(* IEC 61131-3 sources: ics/BLR1_PhoenixContact/BLR1_AXC1050_21/LogicalPOUs/MB, 7 files *)

(* ---- DW_TO_DWORD.ST ---- *)
(*@PROPERTIES_EX@
TYPE: POU
LOCALE: 0
IEC_LANGUAGE: ST
PLC_TYPE: independent
PROC_TYPE: independent
GROUP: MB.FB
*)
(*@KEY@:DESCRIPTION*)

(*@KEY@:END_DESCRIPTION*)
FUNCTION DW_TO_DWORD:DWORD

(*Group:Default*)

VAR_INPUT
    LO_WORD :	WORD;
    HI_WORD :	WORD;
END_VAR

VAR
    OUT_DWORD :	DWORD;
END_VAR

(*@KEY@: WORKSHEET
NAME: DW_TO_DWORD
IEC_LANGUAGE: ST
*)
OUT_DWORD.W0:=HI_WORD;
OUT_DWORD.W1:=LO_WORD;
DW_TO_DWORD:=OUT_DWORD;

(*@KEY@: END_WORKSHEET *)
END_FUNCTION

(* ---- MB_TO_REAL.ST ---- *)
(*@PROPERTIES_EX@
TYPE: POU
LOCALE: 0
IEC_LANGUAGE: ST
PLC_TYPE: independent
PROC_TYPE: independent
GROUP: MB.FB
*)
(*@KEY@:DESCRIPTION*)

(*@KEY@:END_DESCRIPTION*)
FUNCTION_BLOCK MB_TO_REAL

(*Group:Default*)

VAR_INPUT
	LoWord :	WORD;
	HiWord :	WORD;
END_VAR

VAR
	SYS_IEEE_ToReal_1_1 :	SYS_IEEE_ToReal_1;
END_VAR

VAR_OUTPUT
	OUT :	REAL;
END_VAR

VAR
	IEEE :	SYS_ARR_B_1_4;
END_VAR

(*@KEY@: WORKSHEET
NAME: MB_TO_REAL
IEC_LANGUAGE: ST
*)

IEEE[1]:= LoWord.B0;
IEEE[2]:= LoWord.B1;
IEEE[3]:= HiWord.B0;
IEEE[4]:= HiWord.B1;

SYS_IEEE_ToReal_1_1(arrIEEE_Float:= IEEE);
OUT:=SYS_IEEE_ToReal_1_1.rValue;

(*@KEY@: END_WORKSHEET *)
END_FUNCTION_BLOCK

(* ---- MB_TO_REAL_1.ST ---- *)
(*@PROPERTIES_EX@
TYPE: POU
LOCALE: 0
IEC_LANGUAGE: ST
PLC_TYPE: independent
PROC_TYPE: independent
GROUP: MB.FB
*)
(*@KEY@:DESCRIPTION*)

(*@KEY@:END_DESCRIPTION*)
FUNCTION_BLOCK MB_TO_REAL_1

(*Group:Default*)

VAR_INPUT
	LoWord :	WORD;
	HiWord :	WORD;
END_VAR

VAR
	SYS_IEEE_ToReal_1_1 :	SYS_IEEE_ToReal_1;
END_VAR

VAR_OUTPUT
	OUT :	REAL;
END_VAR

VAR
	IEEE :	SYS_ARR_B_1_4;
END_VAR

(*@KEY@: WORKSHEET
NAME: MB_TO_REAL_1
IEC_LANGUAGE: ST
*)

IEEE[1]:= LoWord.B1;
IEEE[2]:= LoWord.B0;
IEEE[3]:= HiWord.B1;
IEEE[4]:= HiWord.B0;

SYS_IEEE_ToReal_1_1(arrIEEE_Float:= IEEE);
OUT:=SYS_IEEE_ToReal_1_1.rValue;

(*@KEY@: END_WORKSHEET *)
END_FUNCTION_BLOCK

(* ---- REAL_TO_MB.ST ---- *)
(*@PROPERTIES_EX@
TYPE: POU
LOCALE: 0
IEC_LANGUAGE: ST
PLC_TYPE: independent
PROC_TYPE: independent
GROUP: MB.FB
*)
(*@KEY@:DESCRIPTION*)

(*@KEY@:END_DESCRIPTION*)
FUNCTION_BLOCK REAL_TO_MB

(*Group:Default*)

VAR_OUTPUT
	LoWord :	WORD;
	HiWord :	WORD;
END_VAR

VAR_INPUT
	IN :	REAL;
END_VAR

VAR
	SYS_RealTo_IEEE_1_1 :	SYS_RealTo_IEEE_1;
	IEEE :	SYS_ARR_B_1_4;
END_VAR

(*@KEY@: WORKSHEET
NAME: REAL_TO_MB
IEC_LANGUAGE: ST
*)

SYS_RealTo_IEEE_1_1(rValue:=IN);
IEEE:=SYS_RealTo_IEEE_1_1.arrIEEE_Float;

LoWord.B0:= IEEE[1];
LoWord.B1:= IEEE[2];
HiWord.B0:= IEEE[3];
HiWord.B1:= IEEE[4];
(*@KEY@: END_WORKSHEET *)
END_FUNCTION_BLOCK

(* ---- MB_RTU_1.ST ---- *)
(*@PROPERTIES_EX@
TYPE: POU
LOCALE: 0
IEC_LANGUAGE: ST
PLC_TYPE: independent
PROC_TYPE: independent
GROUP: MB
*)
(*@KEY@:DESCRIPTION*)

(*@KEY@:END_DESCRIPTION*)
PROGRAM MB_RTU_1

(*Group:NewGroup*)

VAR
    TON_MB_RTU_Master_Startup :	TON;
    MB_AXL_RS_UNI_Act :	BOOL;
    MB_RTU_Master_Act :	BOOL;
    MB_RTU_FC_Act :	BOOL;
    MB_AXL_RS_UNI_REC_2_1 :	MB_AXL_RS_UNI_REC_2;
    udtSerialIF :	MB2_AXL_RSUNI2_UDT_IF;
END_VAR

VAR_EXTERNAL
    arrInData_AXL_RSUNI_1 :	MB2_AXL_RSUNI2_ARR_B_0_19;
    arrOutData_AXL_RSUNI_1 :	MB2_AXL_RSUNI2_ARR_B_0_19;
END_VAR

VAR
    udtDiag_AXL_RSUNI_REC :	MB_UDT_RTU_REC_DIAG;
    wDiagCode_AXL_RSUNI_REC :	WORD;
    wAddDiagCode_AXL_RSUNI_REC :	WORD;
    xError_AXL_RSUNI_REC :	BOOL;
    xBusy_AXL_RSUNI_REC :	BOOL;
    xActive_AXL_RSUNI_REC :	BOOL;
    MB_AXL_RS_UNI_SND_2_1 :	MB_AXL_RS_UNI_SND_2;
    udtDiag_AXL_RSUNI_SND :	MB_UDT_RTU_SND_DIAG;
    wAddDiagCode_AXL_RSUNI_SND :	WORD;
    wDiagCode_AXL_RSUNI_SND :	WORD;
    xError_AXL_RSUNI_SND :	BOOL;
    xBusy_AXL_RSUNI_SND :	BOOL;
    xActive_AXL_RSUNI_SND :	BOOL;
    MB_RTU_Master_4_1 :	MB_RTU_Master_4;
    udtMbData :	udtModbus2_Data;
    udtDiag_RTU_Master :	MB_UDT_RTU_MASTER_DIAG;
    wAddDiagCode_RTU_Master :	WORD;
    wDiagCode_RTU_Master :	WORD;
    xError_RTU_Master :	BOOL;
    xBusy_RTU_Master :	BOOL;
    xActive_RTU_Master :	BOOL;
    uiRespCount_RTU_Master :	UINT;
    uiReqCount_RTU_Master :	UINT;
    MB_RTU_FC3 :	MB_RTU_FC3_3;
    SlvAddr :	MBRTU_SlvAddr;
    RegAddr :	MBRTU_RegAddr;
    arrReadData_RTU_FC3 :	arrModbus2_W_1_125;
    udtDiag_RTU_FC3 :	MB_UDT_RTU_FC_DIAG;
    wAddDiagCode_RTU_FC3 :	WORD;
    wDiagCode_RTU_FC3 :	WORD;
    xError_RTU_FC3 :	BOOL;
    xDone_RTU_FC3 :	BOOL;
    xBusy_RTU_FC3 :	BOOL;
    xActive_RTU_FC3 :	BOOL;
    R_TRIG_1 :	R_TRIG;
    F_TRIG_3 :	F_TRIG;
    i :	INT;
    j :	INT;
    a :	INT;
    b :	INT;
    i1 :	INT;
    State :	INT;
    xSndReq_RTU_FC3 :	BOOL;
END_VAR

VAR_EXTERNAL
    SlvData_RSUNI_1 :	MBRTU_SlvData;
    PLCMODE_RUN :	BOOL;(*PLC status RUN*)
END_VAR

(*@KEY@: WORKSHEET
NAME: MB_RTU_1
IEC_LANGUAGE: ST
*)
(*============================================================================*)
(*MB RTU startup timer*)
(*============================================================================*)
TON_MB_RTU_Master_Startup(IN:= PLCMODE_RUN,PT:=t#2s);
IF TON_MB_RTU_Master_Startup.Q and not (xError_AXL_RSUNI_REC or
    xError_RTU_Master or xError_AXL_RSUNI_SND) THEN
    MB_AXL_RS_UNI_Act		:= true;
    MB_RTU_Master_Act		:= true;
    MB_RTU_FC_Act			:= true;
ELSE
    MB_AXL_RS_UNI_Act		:= false;
    MB_RTU_Master_Act		:= false;
    MB_RTU_FC_Act			:= false;
END_IF;

(*============================================================================*)
(*MB_AXL_UNI_REC FB initialization*)
(*============================================================================*)
MB_AXL_RS_UNI_REC_2_1(xActivate:= MB_AXL_RS_UNI_Act,
    udtSerialIF:= udtSerialIF,
    arrInputData:= arrInData_AXL_RSUNI_1,
    arrOutputData:= arrOutData_AXL_RSUNI_1);

xActive_AXL_RSUNI_REC		:=MB_AXL_RS_UNI_REC_2_1.xActive;
xBusy_AXL_RSUNI_REC			:=MB_AXL_RS_UNI_REC_2_1.xBusy;
xError_AXL_RSUNI_REC		:=MB_AXL_RS_UNI_REC_2_1.xError;
wDiagCode_AXL_RSUNI_REC		:=MB_AXL_RS_UNI_REC_2_1.wDiagCode;
wAddDiagCode_AXL_RSUNI_REC	:=MB_AXL_RS_UNI_REC_2_1.wAddDiagCode;
udtDiag_AXL_RSUNI_REC		:=MB_AXL_RS_UNI_REC_2_1.udtDiag;
udtSerialIF					:=MB_AXL_RS_UNI_REC_2_1.udtSerialIF;
arrInData_AXL_RSUNI_1		:=MB_AXL_RS_UNI_REC_2_1.arrInputData;
arrOutData_AXL_RSUNI_1		:=MB_AXL_RS_UNI_REC_2_1.arrOutputData;

(*============================================================================*)
(*MB RTU Master FB initialization*)
(*============================================================================*)
MB_RTU_Master_4_1(xActivate:= xActive_AXL_RSUNI_REC and xActive_AXL_RSUNI_SND,
    xReset:= false,
    xAuto_CRC:= false,
    tTimeout:= t#200ms,
    udtSerialIF:= udtSerialIF,
    udtMbData:= udtMbData);

xActive_RTU_Master			:=MB_RTU_Master_4_1.xActive;
xBusy_RTU_Master			:=MB_RTU_Master_4_1.xBusy;
uiReqCount_RTU_Master		:=MB_RTU_Master_4_1.uiRequestsCounter;
uiRespCount_RTU_Master		:=MB_RTU_Master_4_1.uiResponsesCounter;
xError_RTU_Master			:=MB_RTU_Master_4_1.xError;
wDiagCode_RTU_Master		:=MB_RTU_Master_4_1.wDiagCode;
wAddDiagCode_RTU_Master		:=MB_RTU_Master_4_1.wAddDiagCode;
udtDiag_RTU_Master			:=MB_RTU_Master_4_1.udtDiag;
udtSerialIF					:=MB_RTU_Master_4_1.udtSerialIF;
udtMbData					:=MB_RTU_Master_4_1.udtMbData;

(*============================================================================*)
(*MB_AXL_UNI_SND FB initialization*)
(*============================================================================*)
MB_AXL_RS_UNI_SND_2_1(xActivate:= MB_AXL_RS_UNI_Act,
    udtSerialIF:= udtSerialIF,
    arrInputData:= arrInData_AXL_RSUNI_1,
    arrOutputData:= arrOutData_AXL_RSUNI_1);

xActive_AXL_RSUNI_SND		:=MB_AXL_RS_UNI_SND_2_1.xActive;
xBusy_AXL_RSUNI_SND			:=MB_AXL_RS_UNI_SND_2_1.xBusy;
xError_AXL_RSUNI_SND		:=MB_AXL_RS_UNI_SND_2_1.xError;
wDiagCode_AXL_RSUNI_SND		:=MB_AXL_RS_UNI_SND_2_1.wDiagCode;
wAddDiagCode_AXL_RSUNI_SND	:=MB_AXL_RS_UNI_SND_2_1.wAddDiagCode;
udtDiag_AXL_RSUNI_SND		:=MB_AXL_RS_UNI_SND_2_1.udtDiag;
udtSerialIF					:=MB_AXL_RS_UNI_SND_2_1.udtSerialIF;
arrInData_AXL_RSUNI_1		:=MB_AXL_RS_UNI_SND_2_1.arrInputData;
arrOutData_AXL_RSUNI_1		:=MB_AXL_RS_UNI_SND_2_1.arrOutputData;

(*============================================================================*)
(*Slaves registers addresses assigning*)
(*============================================================================*)
R_TRIG_1(CLK:= xActive_RTU_Master);

SlvAddr[0]					:= uint#10;                                         (*Pump 5.1 FC MB address*)
SlvAddr[1]					:= uint#11;                                         (*Pump 5.2 FC MB address*)
SlvAddr[2]					:= uint#12;                                         (*Pump 5.3 FC MB address*)

IF R_TRIG_1.Q THEN
    i:= 0;
    j:= 0;
    FOR i1:= 0 to 2 DO
        RegAddr[i1][0]		:= uint#16129;                                      (*reg.16129 Frequency Hz*)
        RegAddr[i1][1]		:= uint#16099;                                      (*reg.16099 Power kWt*)
        RegAddr[i1][2]		:= uint#16139;                                      (*reg.16139 Motor Current A*)
        RegAddr[i1][3]		:= uint#16339;                                      (*reg.16339 HeatSink Temp.*)
        RegAddr[i1][4]		:= uint#16029;                                      (*reg.16029 Status Word*)
        RegAddr[i1][5]		:= uint#16899;                                      (*reg.16899 Alarm Word*)
        RegAddr[i1][6]		:= uint#16919;                                      (*reg.16919 Warning Word*)
        RegAddr[i1][7]		:= uint#15009;                                      (*reg.15009 Running hours h*)
        RegAddr[i1][8]		:= uint#15019;                                      (*reg.15019 kWh Counter*)
    END_FOR;
END_IF;

(*============================================================================*)
(*Pumps FCs parameters reading*)
(*============================================================================*)
MB_RTU_FC3(xActivate:= MB_RTU_Master_Act,
    xSendRequest:= xSndReq_RTU_FC3,
    xEnablePoll:= false,
    tPollInterval:= t#100ms,
    uiSlaveAddress:= SlvAddr[i],
    uiStartAddress:=RegAddr[i][j],
    iDataCount:= 2,
    arrReadData:= arrReadData_RTU_FC3,
    udtMbData:= udtMbData);

xActive_RTU_FC3				:=MB_RTU_FC3.xActive;
xBusy_RTU_FC3				:=MB_RTU_FC3.xBusy;
xDone_RTU_FC3				:=MB_RTU_FC3.xDone;
xError_RTU_FC3				:=MB_RTU_FC3.xError;
wDiagCode_RTU_FC3			:=MB_RTU_FC3.wDiagCode;
wAddDiagCode_RTU_FC3		:=MB_RTU_FC3.wAddDiagCode;
udtDiag_RTU_FC3				:=MB_RTU_FC3.udtDiag;
arrReadData_RTU_FC3			:=MB_RTU_FC3.arrReadData;
udtMbData					:=MB_RTU_FC3.udtMbData;

CASE State OF
    0:
        IF xActive_RTU_Master THEN
            xSndReq_RTU_FC3 := true;
            State:= 10;
        END_IF;

    10:
        IF MB_RTU_FC3.xDone or MB_RTU_FC3.xError THEN
            xSndReq_RTU_FC3 := false;
            State:= 100;
        END_IF;

    100:
        a:= j * 2;
        b:= a + 1;

        SlvData_RSUNI_1[i][a]:= arrReadData_RTU_FC3[1];
        SlvData_RSUNI_1[i][b]:= arrReadData_RTU_FC3[2];
        State:= 1000;

    1000:
        j:= j + 1;
        IF j > 8 THEN
            j:= 0;
            i:= i + 1;
        END_IF;

        IF i > 2 THEN
            i:= 0;
        END_IF;

        State:= 0;
END_CASE;

(*@KEY@: END_WORKSHEET *)
END_PROGRAM

(* ---- MB_RTU_2.ST ---- *)
(*@PROPERTIES_EX@
TYPE: POU
LOCALE: 0
IEC_LANGUAGE: ST
PLC_TYPE: independent
PROC_TYPE: independent
GROUP: MB
*)
(*@KEY@:DESCRIPTION*)

(*@KEY@:END_DESCRIPTION*)
PROGRAM MB_RTU_2

(*Group:NewGroup*)

VAR
	TON_MB_RTU_Master_Startup :	TON;
	MB_AXL_RS_UNI_Act :	BOOL;
	MB_RTU_Master_Act :	BOOL;
	MB_RTU_FC_Act :	BOOL;
	MB_AXL_RS_UNI_REC_2_1 :	MB_AXL_RS_UNI_REC_2;
	udtSerialIF :	MB2_AXL_RSUNI2_UDT_IF;
END_VAR

VAR_EXTERNAL
	arrInData_AXL_RSUNI_2 :	MB2_AXL_RSUNI2_ARR_B_0_19;
	arrOutData_AXL_RSUNI_2 :	MB2_AXL_RSUNI2_ARR_B_0_19;
END_VAR

VAR
	udtDiag_AXL_RSUNI_REC :	MB_UDT_RTU_REC_DIAG;
	wDiagCode_AXL_RSUNI_REC :	WORD;
	wAddDiagCode_AXL_RSUNI_REC :	WORD;
	xError_AXL_RSUNI_REC :	BOOL;
	xBusy_AXL_RSUNI_REC :	BOOL;
	xActive_AXL_RSUNI_REC :	BOOL;
	MB_AXL_RS_UNI_SND_2_1 :	MB_AXL_RS_UNI_SND_2;
	udtDiag_AXL_RSUNI_SND :	MB_UDT_RTU_SND_DIAG;
	wAddDiagCode_AXL_RSUNI_SND :	WORD;
	wDiagCode_AXL_RSUNI_SND :	WORD;
	xError_AXL_RSUNI_SND :	BOOL;
	xBusy_AXL_RSUNI_SND :	BOOL;
	xActive_AXL_RSUNI_SND :	BOOL;
	MB_RTU_Master_4_1 :	MB_RTU_Master_4;
	udtMbData :	udtModbus2_Data;
	udtDiag_RTU_Master :	MB_UDT_RTU_MASTER_DIAG;
	wAddDiagCode_RTU_Master :	WORD;
	wDiagCode_RTU_Master :	WORD;
	xError_RTU_Master :	BOOL;
	xBusy_RTU_Master :	BOOL;
	xActive_RTU_Master :	BOOL;
	uiRespCount_RTU_Master :	UINT;
	uiReqCount_RTU_Master :	UINT;
	MB_RTU_FC3 :	MB_RTU_FC3_3;
	SlvAddr :	MBRTU_SlvAddr;
	RegAddr :	MBRTU_RegAddr;
	arrReadData_RTU_FC3 :	arrModbus2_W_1_125;
	udtDiag_RTU_FC3 :	MB_UDT_RTU_FC_DIAG;
	wAddDiagCode_RTU_FC3 :	WORD;
	wDiagCode_RTU_FC3 :	WORD;
	xError_RTU_FC3 :	BOOL;
	xDone_RTU_FC3 :	BOOL;
	xBusy_RTU_FC3 :	BOOL;
	xActive_RTU_FC3 :	BOOL;
	R_TRIG_1 :	R_TRIG;
	F_TRIG_3 :	F_TRIG;
	i :	INT;
	j :	INT;
	a :	INT;
	State :	INT;
	xSndReq_RTU_FC3 :	BOOL;
	b :	INT;
END_VAR

VAR_EXTERNAL
	SlvData_RSUNI_2 :	MBRTU_SlvData;
END_VAR

VAR
	i1 :	INT;
END_VAR

VAR_EXTERNAL
	PLCMODE_RUN :	BOOL;(*PLC status RUN*)
END_VAR

VAR
	FLG :	BOOL;
END_VAR

(*@KEY@: WORKSHEET
NAME: MB_RTU_2
IEC_LANGUAGE: ST
*)
(*============================================================================*)
(*MB RTU startup timer*)
(*============================================================================*)
TON_MB_RTU_Master_Startup(IN:=PLCMODE_RUN,PT:=t#2s);
IF TON_MB_RTU_Master_Startup.Q and not (xError_AXL_RSUNI_REC or xError_RTU_Master
	or xError_AXL_RSUNI_SND) THEN
	MB_AXL_RS_UNI_Act		:= true;
	MB_RTU_Master_Act		:= true;
	MB_RTU_FC_Act			:= true;
ELSE
	MB_AXL_RS_UNI_Act		:= false;
	MB_RTU_Master_Act		:= false;
	MB_RTU_FC_Act			:= false;
END_IF;

(*============================================================================*)
(*MB_AXL_UNI_REC FB initialization*)
(*============================================================================*)
MB_AXL_RS_UNI_REC_2_1(xActivate:= MB_AXL_RS_UNI_Act,
	udtSerialIF:= udtSerialIF,
	arrInputData:= arrInData_AXL_RSUNI_2,
	arrOutputData:= arrOutData_AXL_RSUNI_2);

xActive_AXL_RSUNI_REC		:=MB_AXL_RS_UNI_REC_2_1.xActive;
xBusy_AXL_RSUNI_REC			:=MB_AXL_RS_UNI_REC_2_1.xBusy;
xError_AXL_RSUNI_REC		:=MB_AXL_RS_UNI_REC_2_1.xError;
wDiagCode_AXL_RSUNI_REC		:=MB_AXL_RS_UNI_REC_2_1.wDiagCode;
wAddDiagCode_AXL_RSUNI_REC	:=MB_AXL_RS_UNI_REC_2_1.wAddDiagCode;
udtDiag_AXL_RSUNI_REC		:=MB_AXL_RS_UNI_REC_2_1.udtDiag;
udtSerialIF					:=MB_AXL_RS_UNI_REC_2_1.udtSerialIF;
arrInData_AXL_RSUNI_2		:=MB_AXL_RS_UNI_REC_2_1.arrInputData;
arrOutData_AXL_RSUNI_2		:=MB_AXL_RS_UNI_REC_2_1.arrOutputData;

(*============================================================================*)
(*MB RTU Master FB initialization*)
(*============================================================================*)
MB_RTU_Master_4_1(xActivate:= xActive_AXL_RSUNI_REC and xActive_AXL_RSUNI_SND,
	xReset:= false,
	xAuto_CRC:= false,
	tTimeout:= t#200ms,
	udtSerialIF:= udtSerialIF,
	udtMbData:= udtMbData);

xActive_RTU_Master			:=MB_RTU_Master_4_1.xActive;
xBusy_RTU_Master			:=MB_RTU_Master_4_1.xBusy;
uiReqCount_RTU_Master		:=MB_RTU_Master_4_1.uiRequestsCounter;
uiRespCount_RTU_Master		:=MB_RTU_Master_4_1.uiResponsesCounter;
xError_RTU_Master			:=MB_RTU_Master_4_1.xError;
wDiagCode_RTU_Master		:=MB_RTU_Master_4_1.wDiagCode;
wAddDiagCode_RTU_Master		:=MB_RTU_Master_4_1.wAddDiagCode;
udtDiag_RTU_Master			:=MB_RTU_Master_4_1.udtDiag;
udtSerialIF					:=MB_RTU_Master_4_1.udtSerialIF;
udtMbData					:=MB_RTU_Master_4_1.udtMbData;

(*============================================================================*)
(*MB_AXL_UNI_SND FB initialization*)
(*============================================================================*)
MB_AXL_RS_UNI_SND_2_1(xActivate:= MB_AXL_RS_UNI_Act,
	udtSerialIF:= udtSerialIF,
	arrInputData:= arrInData_AXL_RSUNI_2,
	arrOutputData:= arrOutData_AXL_RSUNI_2);

xActive_AXL_RSUNI_SND		:=MB_AXL_RS_UNI_SND_2_1.xActive;
xBusy_AXL_RSUNI_SND			:=MB_AXL_RS_UNI_SND_2_1.xBusy;
xError_AXL_RSUNI_SND		:=MB_AXL_RS_UNI_SND_2_1.xError;
wDiagCode_AXL_RSUNI_SND		:=MB_AXL_RS_UNI_SND_2_1.wDiagCode;
wAddDiagCode_AXL_RSUNI_SND	:=MB_AXL_RS_UNI_SND_2_1.wAddDiagCode;
udtDiag_AXL_RSUNI_SND		:=MB_AXL_RS_UNI_SND_2_1.udtDiag;
udtSerialIF					:=MB_AXL_RS_UNI_SND_2_1.udtSerialIF;
arrInData_AXL_RSUNI_2		:=MB_AXL_RS_UNI_SND_2_1.arrInputData;
arrOutData_AXL_RSUNI_2		:=MB_AXL_RS_UNI_SND_2_1.arrOutputData;

(*============================================================================*)
(*Slaves registers addresses assigning*)
(*============================================================================*)
R_TRIG_1(CLK:= xActive_RTU_Master);

SlvAddr[0]					:= uint#10;											(*Pump 3.1 FC MB address*)
SlvAddr[1]					:= uint#11;											(*Pump 3.2 FC MB address*)
SlvAddr[2]					:= uint#12;											(*Pump 3.3 FC MB address*)
SlvAddr[3]					:= uint#13;											(*Pump 6.1 FC MB address*)
SlvAddr[4]					:= uint#14;											(*Pump 6.2 FC MB address*)

SlvAddr[5]					:= uint#21;											(*FT020 MB address*)
SlvAddr[6]					:= uint#22;											(*FT1107 MB address*)
SlvAddr[7]					:= uint#23;											(*FT1207 MB address*)
SlvAddr[8]					:= uint#24;											(*FT1307 MB address*)
SlvAddr[9]					:= uint#25;											(*FT2108 MB address*)
SlvAddr[10]					:= uint#20;											(*FT2208 MB address*)

IF R_TRIG_1.Q or FLG THEN
	i:= 0;
	j:= 0;
	FOR i1:= 0 to 4 DO
		RegAddr[i1][0]		:= uint#16129;										(*reg.16129 Frequency Hz*)
		RegAddr[i1][1]		:= uint#16099;										(*reg.16099 Power kWt*)
		RegAddr[i1][2]		:= uint#16139;										(*reg.16139 Motor Current A*)
		RegAddr[i1][3]		:= uint#16339;										(*reg.16339 HeatSink Temp.*)
		RegAddr[i1][4]		:= uint#16029;										(*reg.16029 Status Word*)
		RegAddr[i1][5]		:= uint#16899;										(*reg.16899 Alarm Word*)
		RegAddr[i1][6]		:= uint#16919;										(*reg.16919 Warning Word*)
		RegAddr[i1][7]		:= uint#15009;										(*reg.15009 Running hours h*)
		RegAddr[i1][8]		:= uint#15019;										(*reg.15019 kWh Counter*)
	END_FOR;

	FOR i1:= 5 to 9 DO
		RegAddr[i1][0]		:= uint#3874;										(*reg.3874 Volume flow*)
		RegAddr[i1][1]		:= uint#2610;										(*reg.2610 Totalizer val.*)
	END_FOR;

		RegAddr[10][0]		:= uint#0;											(*reg.0 Volume flow*)
		RegAddr[10][1]		:= uint#2;											(*reg.2 Totalizer val.*)

END_IF;

(*============================================================================*)
(*Pumps FCs parameters reading*)
(*============================================================================*)
MB_RTU_FC3(xActivate:= MB_RTU_Master_Act,
	xSendRequest:= xSndReq_RTU_FC3,
	xEnablePoll:=false,
	tPollInterval:= t#100ms,
	uiSlaveAddress:= SlvAddr[i],
	uiStartAddress:=RegAddr[i][j],
	iDataCount:= 2,
	arrReadData:= arrReadData_RTU_FC3,
	udtMbData:= udtMbData);

xActive_RTU_FC3				:=MB_RTU_FC3.xActive;
xBusy_RTU_FC3				:=MB_RTU_FC3.xBusy;
xDone_RTU_FC3				:=MB_RTU_FC3.xDone;
xError_RTU_FC3				:=MB_RTU_FC3.xError;
wDiagCode_RTU_FC3			:=MB_RTU_FC3.wDiagCode;
wAddDiagCode_RTU_FC3		:=MB_RTU_FC3.wAddDiagCode;
udtDiag_RTU_FC3				:=MB_RTU_FC3.udtDiag;
arrReadData_RTU_FC3			:=MB_RTU_FC3.arrReadData;
udtMbData					:=MB_RTU_FC3.udtMbData;

CASE State OF
	0:
		IF xActive_RTU_Master THEN
			xSndReq_RTU_FC3 := true;
			State:= 10;
		END_IF;

	10:
		IF MB_RTU_FC3.xDone or MB_RTU_FC3.xError THEN
			xSndReq_RTU_FC3 := false;
			State:= 100;
		END_IF;

	100:
		a:= j * 2;
		b:= a + 1;

		SlvData_RSUNI_2[i][a]:= arrReadData_RTU_FC3[1];
		SlvData_RSUNI_2[i][b]:= arrReadData_RTU_FC3[2];
		State:= 1000;

	1000:
		j:= j + 1;
		IF (j > 8) or ((i > 4) and (j > 1)) THEN
			j:= 0;
			i:= i + 1;
		END_IF;

		IF i > 10 THEN
			i:= 0;
		END_IF;

		State:= 0;
END_CASE;

(*@KEY@: END_WORKSHEET *)
END_PROGRAM

(* ---- MB_TCP.ST ---- *)
(*@PROPERTIES_EX@
TYPE: POU
LOCALE: 0
IEC_LANGUAGE: ST
PLC_TYPE: independent
PROC_TYPE: independent
GROUP: MB
*)
(*@KEY@:DESCRIPTION*)

(*@KEY@:END_DESCRIPTION*)
PROGRAM MB_TCP

(*Group:Default*)

VAR
	TON_MBTCP_Master_Startup :	TON;
END_VAR

VAR_EXTERNAL
	PLCMODE_RUN :	BOOL;(*PLC status RUN*)
END_VAR

VAR
	MBTCP_SrvAct :	BOOL;
	MBTCP_Srv1Err :	BOOL;
	MB_TCP_Server_1 :	MB_TCP_Server_1;
	MBTCP_Srv1Ack :	BOOL;
END_VAR

VAR_EXTERNAL
	MBTCP_Data :	MB_TCP_ARR_W_0_7167;
END_VAR

VAR
	MBTCP_Srv1Active :	BOOL;
	MBTCP_Srv1Conn :	BOOL;
	MBTCP_Srv1DiagCode :	WORD;
	MBTCP_Srv1AddDiagCode :	WORD;
	MBTCP_Srv1Diag :	MB_TCP_UDT_SER_DIAG;
	MBTCP_Srv2Active :	BOOL;
	MBTCP_Srv2Conn :	BOOL;
	MBTCP_Srv2Err :	BOOL;
	MBTCP_Srv2DiagCode :	WORD;
	MBTCP_Srv2AddDiagCode :	WORD;
	MBTCP_Srv2Diag :	MB_TCP_UDT_SER_DIAG;
END_VAR

VAR_EXTERNAL
	AI :	SENSOR;
END_VAR

VAR
	i :	INT;
	j :	INT;
	j1 :	INT;
	j2 :	INT;
	j3 :	INT;
	j4 :	INT;
	j5 :	INT;
	j6 :	INT;
	j7 :	INT;
	j8 :	INT;
	j9 :	INT;
	j10 :	INT;
	j11 :	INT;
	j12 :	INT;
	j13 :	INT;
	j14 :	INT;
	j15 :	INT;
	j16 :	INT;
	j17 :	INT;
	j18 :	INT;
	j19 :	INT;
	j20 :	INT;
	j21 :	INT;
	j22 :	INT;
	j23 :	INT;
	j24 :	INT;
	j25 :	INT;
	j26 :	INT;
	j27 :	INT;
	j28 :	INT;
	j29 :	INT;
	j30 :	INT;
	j31 :	INT;
	MB_TO_REAL :	MB_TO_REAL;
	REAL_TO_MB :	REAL_TO_MB;
END_VAR

VAR_EXTERNAL
	M :	MOTOR;
END_VAR

VAR
	MB_TCP_Server_2 :	MB_TCP_Server_1;
END_VAR

VAR_EXTERNAL
	V :	VALVE;
	RGLTR :	REGULATOR;
	CCL :	CYCLE;
	M_AUX :	MOTOR_MISC;
END_VAR

VAR
	MB_TCP_Server :	MB_TCP_Server_1;
	MBTCP_SrvActive :	BOOL;
	MBTCP_SrvConn :	BOOL;
	MBTCP_SrvErr :	BOOL;
	MBTCP_SrvDiagCode :	WORD;
	MBTCP_SrvAddDiagCode :	WORD;
	MBTCP_SrvDiag :	MB_TCP_UDT_SER_DIAG;
	MBTCP_DataScd :	MB_TCP_ARR_W_0_7167;
	MBTCP_SrvAck :	BOOL;
END_VAR

(*@KEY@: WORKSHEET
NAME: MB_TCP
IEC_LANGUAGE: ST
*)
(*============================================================================*)
(*MB TCP startup timer*)
(*============================================================================*)
TON_MBTCP_Master_Startup(IN:=PLCMODE_RUN,PT:=t#2s);
MBTCP_SrvAct:= TON_MBTCP_Master_Startup.Q;

(*============================================================================*)
(*MB TCP server FB initialization port 502*)
(*============================================================================*)
MB_TCP_Server(xActivate:=MBTCP_SrvAct,
	xAcknowledge:=MBTCP_SrvAck,
	xAutoAck:=true,
	xUDP_Mode:=false,
	iTCP_Port:=502,
	(*strPartner_IP:= STRING *)
	tReconnectDelay:=t#100ms,
	tTimeout:=t#0s,
	uiOffsetInputRegister:=uint#0,
	uiOffsetHoldingRegister:=uint#0,
	uiOffsetInputs:=uint#0,
	uiOffsetCoils:=uint#0,
	arrModbusData:=MBTCP_DataScd);

	MBTCP_SrvActive:=MB_TCP_Server.xActive;
	MBTCP_SrvConn:=MB_TCP_Server.xConnected;
	MBTCP_SrvErr:=MB_TCP_Server.xError;
	MBTCP_SrvDiagCode:=MB_TCP_Server.wDiagCode;
	MBTCP_SrvAddDiagCode:=MB_TCP_Server.wAddDiagCode;
	MBTCP_SrvDiag:=MB_TCP_Server.udtDiag;
	MBTCP_DataScd:=MB_TCP_Server.arrModbusData;

(*============================================================================*)
(*MB TCP server #1 FB initialization port 503*)
(*============================================================================*)
MB_TCP_Server_1(xActivate:=MBTCP_SrvAct,
	xAcknowledge:=MBTCP_Srv1Ack,
	xAutoAck:=true,
	xUDP_Mode:=false,
	iTCP_Port:=503,
	(*strPartner_IP:= STRING *)
	tReconnectDelay:=t#100ms,
	tTimeout:=t#0s,
	uiOffsetInputRegister:=uint#0,
	uiOffsetHoldingRegister:=uint#0,
	uiOffsetInputs:=uint#0,
	uiOffsetCoils:=uint#0,
	arrModbusData:=MBTCP_Data);

	MBTCP_Srv1Active:=MB_TCP_Server_1.xActive;
	MBTCP_Srv1Conn:=MB_TCP_Server_1.xConnected;
	MBTCP_Srv1Err:=MB_TCP_Server_1.xError;
	MBTCP_Srv1DiagCode:=MB_TCP_Server_1.wDiagCode;
	MBTCP_Srv1AddDiagCode:=MB_TCP_Server_1.wAddDiagCode;
	MBTCP_Srv1Diag:=MB_TCP_Server_1.udtDiag;
	MBTCP_Data:=MB_TCP_Server_1.arrModbusData;

(*============================================================================*)
(*MB TCP server #2 FB initialization port 503*)
(*============================================================================*)
MB_TCP_Server_2(xActivate:=MBTCP_SrvAct,
	xAcknowledge:=MBTCP_Srv1Ack,
	xAutoAck:=true,
	xUDP_Mode:=false,
	iTCP_Port:=503,
	(*strPartner_IP:= STRING *)
	tReconnectDelay:=t#100ms,
	tTimeout:=t#0s,
	uiOffsetInputRegister:=uint#0,
	uiOffsetHoldingRegister:=uint#0,
	uiOffsetInputs:=uint#0,
	uiOffsetCoils:=uint#0,
	arrModbusData:=MBTCP_Data);

	MBTCP_Srv2Active:=MB_TCP_Server_2.xActive;
	MBTCP_Srv2Conn:=MB_TCP_Server_2.xConnected;
	MBTCP_Srv2Err:=MB_TCP_Server_2.xError;
	MBTCP_Srv2DiagCode:=MB_TCP_Server_2.wDiagCode;
	MBTCP_Srv2AddDiagCode:=MB_TCP_Server_2.wAddDiagCode;
	MBTCP_Srv2Diag:=MB_TCP_Server_2.udtDiag;
	MBTCP_Data:=MB_TCP_Server_2.arrModbusData;

(*============================================================================*)
(*Read/Write cycles data from/to Modbus array  / addr.0 - addr.9*)
(*============================================================================*)
FOR i:= 0 to 4 DO
	j:= i * 2;
	j1:= j + 1;

	CCL[i].CW.Start	:=MBTCP_Data[j].X1;
	CCL[i].CW.Stop:=MBTCP_Data[j].X2;
	CCL[i].CW.ACK:=MBTCP_Data[j].X4;
	CCL[i].CW.Rotation:=MBTCP_Data[j].X8;
	MBTCP_Data[j]:=word#0;

	MBTCP_Data[j1].X0:=CCL[i].SW.ALARM;
	MBTCP_Data[j1].X1:=CCL[i].SW.ON;
	MBTCP_Data[j1].X2:=CCL[i].SW.Running;
	MBTCP_Data[j1].X8:=CCL[i].SW.RotationON;
END_FOR;

(*============================================================================*)
(*Read/Write sensors parameters from/to Modbus array  / addr.100 - addr.3938*)
(*============================================================================*)
FOR i:= 0 to 119 DO
	j:= i * 32 + 100;
	j1:= j + 1;
	j2:= j + 2;
	j3:= j + 3;
	j4:= j + 4;
	j5:= j + 5;
	j6:= j + 6;
	j7:= j + 7;
	j8:= j + 8;
	j9:= j + 9;
	j10:= j + 10;
	j11:= j + 11;
	j12:= j + 12;
	j13:= j + 13;
	j14:= j + 14;
	j15:= j + 15;
	j16:= j + 16;
	j17:= j + 17;
	j18:= j + 18;
	j19:= j + 19;
	j20:= j + 20;
	j21:= j + 21;
	j22:= j + 22;
	j23:= j + 23;
	j24:= j + 24;
	j25:= j + 25;
	j26:= j + 26;
	j27:= j + 27;
	j28:= j + 28;
	j29:= j + 29;
	j30:= j + 30;
	j31:= j + 31;

	AI[i].CW.FltrEn:=MBTCP_Data[j].X0;
	AI[i].CW.LimEn:=MBTCP_Data[j].X1;
	AI[i].CW.SimEn:=MBTCP_Data[j].X2;

	MBTCP_Data[j1].X0:=AI[i].SW.Fault;
	MBTCP_Data[j1].X1:=AI[i].SW.HH_alarm;
	MBTCP_Data[j1].X2:=AI[i].SW.HL_alarm;
	MBTCP_Data[j1].X3:=AI[i].SW.LH_alarm;
	MBTCP_Data[j1].X4:=AI[i].SW.LL_alarm;

	MB_TO_REAL(LoWord:=MBTCP_Data[j2],HiWord:=MBTCP_Data[j3]);
	AI[i].Ymin:=MB_TO_REAL.OUT;

	MB_TO_REAL(LoWord:=MBTCP_Data[j4],HiWord:=MBTCP_Data[j5]);
	AI[i].Ymax:=MB_TO_REAL.OUT;

	(*AI[i].ADC_Range:=word_to_int(MBTCP_Data[j6]);*)
	AI[i].SamplingTime:=word_to_int(MBTCP_Data[j7]);

	MB_TO_REAL(LoWord:=MBTCP_Data[j8],HiWord:=MBTCP_Data[j9]);
	AI[i].HH:=MB_TO_REAL.OUT;

	MB_TO_REAL(LoWord:=MBTCP_Data[j10],HiWord:=MBTCP_Data[j11]);
	AI[i].HL:=MB_TO_REAL.OUT;

	MB_TO_REAL(LoWord:=MBTCP_Data[j12],HiWord:=MBTCP_Data[j13]);
	AI[i].LH:=MB_TO_REAL.OUT;

	MB_TO_REAL(LoWord:=MBTCP_Data[j14],HiWord:=MBTCP_Data[j15]);
	AI[i].LL:=MB_TO_REAL.OUT;

	MB_TO_REAL(LoWord:=MBTCP_Data[j16],HiWord:=MBTCP_Data[j17]);
	AI[i].DeadBand:=MB_TO_REAL.OUT;

	AI[i].LimDelay:=word_to_int(MBTCP_Data[j18]);

	MBTCP_Data[j19]:=AI[i].DiagCode;

(*	MB_TO_REAL(LoWord:=MBTCP_Data[j20],HiWord:=MBTCP_Data[j21]);
	AI[i].res1:=MB_TO_REAL.OUT;	*)

	MBTCP_Data[j22]:=int_to_word(AI[i].PIW);
	MBTCP_Data[j23]:=int_to_word(AI[i].IntValue);

	REAL_TO_MB(IN:=AI[i].RealValue);
	MBTCP_Data[j24]:=REAL_TO_MB.LoWord;
	MBTCP_Data[j25]:=REAL_TO_MB.HiWord;

	MB_TO_REAL(LoWord:=MBTCP_Data[j26],HiWord:=MBTCP_Data[j27]);
	AI[i].SimValue:=MB_TO_REAL.OUT;
END_FOR;

(*============================================================================*)
(*Read/Write motors parameters from/to Modbus array  / addr.3940 - addr.4578*)
(*============================================================================*)
FOR i:= 0 to 19 DO
	j:= i * 32 + 3940;
	j1:= j + 1;
	j2:= j + 2;
	j3:= j + 3;
	j4:= j + 4;
	j5:= j + 5;
	j6:= j + 6;
	j7:= j + 7;
	j8:= j + 8;
	j9:= j + 9;
	j10:= j + 10;
	j11:= j + 11;
	j12:= j + 12;
	j13:= j + 13;
	j14:= j + 14;
	j15:= j + 15;
	j16:= j + 16;
	j17:= j + 17;
	j18:= j + 18;
	j19:= j + 19;
	j20:= j + 20;
	j21:= j + 21;
	j22:= j + 22;
	j23:= j + 23;
	j24:= j + 24;
	j25:= j + 25;
	j26:= j + 26;
	j27:= j + 27;
	j28:= j + 28;
	j29:= j + 29;
	j30:= j + 30;
	j31:= j + 31;

	M[i].CW.ACK:=MBTCP_Data[j].X3;
	M[i].CW.ManMode:=MBTCP_Data[j].X4;
	M[i].CW.AutoMode:=MBTCP_Data[j].X5;
	M[i].CW.ManStart:=MBTCP_Data[j].X6;
	M[i].CW.ManStop:=MBTCP_Data[j].X7;
	M[i].CW.SimEn:=MBTCP_Data[j].X15;
	MBTCP_Data[j]:=word#0;

	MBTCP_Data[j1].X0:=M[i].SW.Rem;
	MBTCP_Data[j1].X1:=M[i].SW.ManAuto;
	MBTCP_Data[j1].X2:=M[i].SW.RUN;
	MBTCP_Data[j1].X3:=M[i].SW.COM;
	MBTCP_Data[j1].X4:=M[i].SW.AlarmAccum;
	MBTCP_Data[j1].X5:=M[i].SW.Ready;

	MB_TO_REAL(LoWord:=MBTCP_Data[j2],HiWord:=MBTCP_Data[j3]);
	M[i].MinFreq:=MB_TO_REAL.OUT;

	MB_TO_REAL(LoWord:=MBTCP_Data[j4],HiWord:=MBTCP_Data[j5]);
	M[i].MaxFreq:=MB_TO_REAL.OUT;

	MB_TO_REAL(LoWord:=MBTCP_Data[j6],HiWord:=MBTCP_Data[j7]);
	M[i].ManFreq:=MB_TO_REAL.OUT;

	REAL_TO_MB(IN:=M[i].ActFreq);
	MBTCP_Data[j10]:=REAL_TO_MB.LoWord;
	MBTCP_Data[j11]:=REAL_TO_MB.HiWord;

	REAL_TO_MB(IN:=M[i].Current);
	MBTCP_Data[j12]:=REAL_TO_MB.LoWord;
	MBTCP_Data[j13]:=REAL_TO_MB.HiWord;

	REAL_TO_MB(IN:=M[i].Power);
	MBTCP_Data[j14]:=REAL_TO_MB.LoWord;
	MBTCP_Data[j15]:=REAL_TO_MB.HiWord;

	REAL_TO_MB(IN:=M[i].HeatSinkTemp);
	MBTCP_Data[j16]:=REAL_TO_MB.LoWord;
	MBTCP_Data[j17]:=REAL_TO_MB.HiWord;

	REAL_TO_MB(IN:=M[i].RunHours);
	MBTCP_Data[j18]:=REAL_TO_MB.LoWord;
	MBTCP_Data[j19]:=REAL_TO_MB.HiWord;

	REAL_TO_MB(IN:=M[i].kWhCount);
	MBTCP_Data[j20]:=REAL_TO_MB.LoWord;
	MBTCP_Data[j21]:=REAL_TO_MB.HiWord;

	MBTCP_Data[j22]:=M[i].Status;
	MBTCP_Data[j23]:=M[i].FC_StatusWord;

	MBTCP_Data[j24]:=M[i].FC_AlarmWord.W0;
	MBTCP_Data[j25]:=M[i].FC_AlarmWord.W1;

	MBTCP_Data[j26]:=M[i].FC_WarnWord.W0;
	MBTCP_Data[j27]:=M[i].FC_WarnWord.W1;

	MBTCP_Data[j28]:=M[i].FC_ErrCode;
	MBTCP_Data[j29]:=M[i].Index;
END_FOR;

(*============================================================================*)
(*Read/Write valves parameters from/to Modbus array  / addr.4580 - addr.4898*)
(*============================================================================*)
FOR i:= 0 to 19 DO
	j:= i * 16 + 4580;
	j1:= j + 1;
	j2:= j + 2;
	j3:= j + 3;
	j4:= j + 4;
	j5:= j + 5;
	j6:= j + 6;
	j7:= j + 7;
	j8:= j + 8;
	j9:= j + 9;
	j10:= j + 10;
	j11:= j + 11;
	j12:= j + 12;
	j13:= j + 13;
	j14:= j + 14;
	j15:= j + 15;

	V[i].CW.ACK	:=MBTCP_Data[j].X3;
	V[i].CW.ManMode:=MBTCP_Data[j].X4;
	V[i].CW.AutoMode:=MBTCP_Data[j].X5;
	V[i].CW.ManOpen:=MBTCP_Data[j].X6;
	V[i].CW.Stop:=MBTCP_Data[j].X7;
	V[i].CW.ManClose:=MBTCP_Data[j].X8;
	V[i].CW.SimEn:=MBTCP_Data[j].X15;
	MBTCP_Data[j]:=word#0;

	MBTCP_Data[j1].X0:=V[i].SW.Rem;
	MBTCP_Data[j1].X1:=V[i].SW.ManAuto;
	MBTCP_Data[j1].X2:=V[i].SW.RUN;
	MBTCP_Data[j1].X3:=V[i].SW.COM_Open;
	MBTCP_Data[j1].X4:=V[i].SW.COM_Close;
	MBTCP_Data[j1].X5:=V[i].SW.Opened;
	MBTCP_Data[j1].X6:=V[i].SW.Closed;
	MBTCP_Data[j1].X7:=V[i].SW.AlarmAccum;

	MB_TO_REAL(LoWord:=MBTCP_Data[j2],HiWord:=MBTCP_Data[j3]);
	V[i].SetPos:=MB_TO_REAL.OUT;

	REAL_TO_MB(IN:=V[i].ActPos);
	MBTCP_Data[j4]:=REAL_TO_MB.LoWord;
	MBTCP_Data[j5]:=REAL_TO_MB.HiWord;

	MBTCP_Data[j6]:=V[i].Status;
END_FOR;

(*============================================================================*)
(*Read/Write regulators parameters from/to Modbus array  / addr.4900 - addr.5538*)
(*============================================================================*)
FOR i:= 0 to 19 DO
	j:= i * 32 + 4900;
	j1:= j + 1;
	j2:= j + 2;
	j3:= j + 3;
	j4:= j + 4;
	j5:= j + 5;
	j6:= j + 6;
	j7:= j + 7;
	j8:= j + 8;
	j9:= j + 9;
	j10:= j + 10;
	j11:= j + 11;
	j12:= j + 12;
	j13:= j + 13;
	j14:= j + 14;
	j15:= j + 15;
	j16:= j + 16;
	j17:= j + 17;
	j18:= j + 18;
	j19:= j + 19;
	j20:= j + 20;
	j21:= j + 21;
	j22:= j + 22;
	j23:= j + 23;
	j24:= j + 24;
	j25:= j + 25;
	j26:= j + 26;
	j27:= j + 27;
	j28:= j + 28;
	j29:= j + 29;
	j30:= j + 30;
	j31:= j + 31;

(*	RGLTR[i].CW.En:=MBTCP_Data[j].X0;
	RGLTR[i].CW.ManMode:=MBTCP_Data[j].X1;
	RGLTR[i].CW.Reset:=MBTCP_Data[j].X2;
	RGLTR[i].CW.Hold:=MBTCP_Data[j].X3;
	RGLTR[i].CW.SimEn:=MBTCP_Data[j].X15;
	MBTCP_Data[j]:=word#0;*)

	MBTCP_Data[j1].X0:=RGLTR[i].SW.Error;
	MBTCP_Data[j1].X1:=RGLTR[i].SW.LH;
	MBTCP_Data[j1].X2:=RGLTR[i].SW.LL;

	MB_TO_REAL(LoWord:=MBTCP_Data[j2],HiWord:=MBTCP_Data[j3]);
	RGLTR[i].SP:=MB_TO_REAL.OUT;

	MB_TO_REAL(LoWord:=MBTCP_Data[j4],HiWord:=MBTCP_Data[j5]);
	RGLTR[i].Kp:=MB_TO_REAL.OUT;

	MB_TO_REAL(LoWord:=MBTCP_Data[j6],HiWord:=MBTCP_Data[j7]);
	RGLTR[i].Tn:=MB_TO_REAL.OUT;

	MB_TO_REAL(LoWord:=MBTCP_Data[j8],HiWord:=MBTCP_Data[j9]);
	RGLTR[i].Tv:=MB_TO_REAL.OUT;

	MB_TO_REAL(LoWord:=MBTCP_Data[j10],HiWord:=MBTCP_Data[j11]);
	RGLTR[i].Td:=MB_TO_REAL.OUT;

	MB_TO_REAL(LoWord:=MBTCP_Data[j12],HiWord:=MBTCP_Data[j13]);
	RGLTR[i].Offset:=MB_TO_REAL.OUT;

	MB_TO_REAL(LoWord:=MBTCP_Data[j14],HiWord:=MBTCP_Data[j15]);
	RGLTR[i].ManVal:=MB_TO_REAL.OUT;

(*	MB_TO_REAL(LoWord:=MBTCP_Data[j16],HiWord:=MBTCP_Data[j17]);
	RGLTR[i].LH:=MB_TO_REAL.OUT;

	MB_TO_REAL(LoWord:=MBTCP_Data[j18],HiWord:=MBTCP_Data[j19]);
	RGLTR[i].LL:=MB_TO_REAL.OUT;*)

	REAL_TO_MB(IN:=RGLTR[i].Y);
	MBTCP_Data[j20]:=REAL_TO_MB.LoWord;
	MBTCP_Data[j21]:=REAL_TO_MB.HiWord;

	REAL_TO_MB(IN:=RGLTR[i].DIFF);
	MBTCP_Data[j22]:=REAL_TO_MB.LoWord;
	MBTCP_Data[j23]:=REAL_TO_MB.HiWord;

	REAL_TO_MB(IN:=RGLTR[i].ActVal);
	MBTCP_Data[j24]:=REAL_TO_MB.LoWord;
	MBTCP_Data[j25]:=REAL_TO_MB.HiWord;

	MB_TO_REAL(LoWord:=MBTCP_Data[j26],HiWord:=MBTCP_Data[j27]);
	RGLTR[i].DeadBand:=MB_TO_REAL.OUT;
END_FOR;

(*============================================================================*)

(*============================================================================*)
(*DATA FOR SCADA*)
(*============================================================================*)
(*============================================================================*)
(*Read/Write 5.x pumps cycle from/to Modbus array  / addr.20 - addr.21*)
(*============================================================================*)
(*	CCL[3].CW.Start:=MBTCP_DataScd[20].X1;
	CCL[3].CW.Stop:=MBTCP_DataScd[20].X2;
	CCL[3].CW.ACK:=MBTCP_DataScd[20].X4;
	CCL[3].CW.Rotation:=MBTCP_DataScd[20].X8;*)

	MBTCP_DataScd[30].X0:=CCL[3].SW.ALARM;
	MBTCP_DataScd[30].X2:=CCL[3].SW.Running;
	MBTCP_DataScd[30].X8:=CCL[3].SW.RotationON;

(*============================================================================*)
(*Read/Write 5.x pumps parameters from/to Modbus array  / addr.100 - addr.189*)
(*============================================================================*)
FOR i:= 8 to 10 DO
	j:= i * 30 - 140;
	j1:= j + 1;
	j2:= j + 2;
	j3:= j + 3;
	j4:= j + 4;
	j5:= j + 5;
	j6:= j + 6;
	j7:= j + 7;
	j8:= j + 8;
	j9:= j + 9;
	j10:= j + 10;
	j11:= j + 11;
	j12:= j + 12;
	j13:= j + 13;
	j14:= j + 14;
	j15:= j + 15;
	j16:= j + 16;
	j17:= j + 17;
	j18:= j + 18;
	j19:= j + 19;
	j20:= j + 20;
	j21:= j + 21;
	j22:= j + 22;
	j23:= j + 23;
	j24:= j + 24;
	j25:= j + 25;
	j26:= j + 26;
	j27:= j + 27;
	j28:= j + 28;
	j29:= j + 29;

(*	M[i].CW.AutoMode:=MBTCP_DataScd[j].X5;
	M[i].CW.ManMode:=MBTCP_DataScd[j].X4;
	M[i].CW.ManStart:=MBTCP_DataScd[j].X6;
	M[i].CW.ManStop:=MBTCP_DataScd[j].X7;
	M[i].CW.ACK:=MBTCP_DataScd[j].X15;*)

	MBTCP_DataScd[j1].X0:=M[i].SW.Rem;
	MBTCP_DataScd[j1].X1:=M[i].SW.ManAuto;
	MBTCP_DataScd[j1].X2:=M[i].SW.RUN;
	MBTCP_DataScd[j1].X3:=M[i].SW.COM;
	MBTCP_DataScd[j1].X4:=M[i].SW.AlarmAccum;

	MB_TO_REAL(LoWord:=MBTCP_DataScd[j2],HiWord:=MBTCP_DataScd[j3]);
	M[i].ManFreq:=MB_TO_REAL.OUT;

	REAL_TO_MB(IN:=M[i].ActFreq);
	MBTCP_DataScd[j4]:=REAL_TO_MB.LoWord;
	MBTCP_DataScd[j5]:=REAL_TO_MB.HiWord;

	MBTCP_DataScd[j6]:=M[i].Status;
	MBTCP_DataScd[j7]:=M[i].Status;

	REAL_TO_MB(IN:=M[i].Current);
	MBTCP_DataScd[j8]:=REAL_TO_MB.LoWord;
	MBTCP_DataScd[j9]:=REAL_TO_MB.HiWord;

	REAL_TO_MB(IN:=M[i].Power);
	MBTCP_DataScd[j10]:=REAL_TO_MB.LoWord;
	MBTCP_DataScd[j11]:=REAL_TO_MB.HiWord;

	REAL_TO_MB(IN:=M[i].HeatSinkTemp);
	MBTCP_DataScd[j12]:=REAL_TO_MB.LoWord;
	MBTCP_DataScd[j13]:=REAL_TO_MB.HiWord;

	REAL_TO_MB(IN:=M[i].RunHours);
	MBTCP_DataScd[j14]:=REAL_TO_MB.LoWord;
	MBTCP_DataScd[j15]:=REAL_TO_MB.HiWord;

	REAL_TO_MB(IN:=M[i].kWhCount);
	MBTCP_DataScd[j16]:=REAL_TO_MB.LoWord;
	MBTCP_DataScd[j17]:=REAL_TO_MB.HiWord;

	MBTCP_DataScd[j18]:=M[i].FC_ErrCode;
END_FOR;

(*============================================================================*)
(*Read/Write 5.x pumps parameters from/to Modbus array  / addr.3002 - addr.xxx*)
(*============================================================================*)
FOR i:= 0 to 5 DO
	j:= i * 2 + 3002;
	j1:= j + 1;

	REAL_TO_MB(IN:=AI[i].RealValue);
	MBTCP_DataScd[j]:=REAL_TO_MB.LoWord;
	MBTCP_DataScd[j1]:=REAL_TO_MB.HiWord;
END_FOR;

MBTCP_DataScd[65].X1:=AI[0].SW.Fault;
MBTCP_DataScd[65].X2:=AI[1].SW.Fault;
MBTCP_DataScd[65].X3:=AI[2].SW.Fault;
MBTCP_DataScd[65].X4:=AI[3].SW.Fault;
MBTCP_DataScd[65].X5:=AI[4].SW.Fault;
MBTCP_DataScd[65].X6:=AI[5].SW.Fault;

(*@KEY@: END_WORKSHEET *)
END_PROGRAM
